// TIA Portal V20 export
TYPE "LER_typeCommonDataInspection"
// stored: Access Published
   STRUCT
      PartType : Byte;   // Part type of jelly roll
      PartStatus : Byte;   // Part status 0: wrong, 1: no part, 2: OK, 3: NOK...
      LastLegNumber : Char;   // Leg no A: stacking #1, B: stacking #2
      LastMachineNumber : Word;   // Last machine no: 20, 30, 60
      ProductionTimestamp : DTL;   // Time of last operation or machining
      Part_ID : String[32];   // Part ID
      ReworkRequested : Bool;   // Request to re-work
   END_STRUCT;
END_TYPE
